FUNCTION_BLOCK TWOCONRINGTOKEN (* Composite Function Block Type *)
  (* Standard: 61499-2 *)
  (* Version 0.2, 2003-12-05, JHC, Rockwell Automation, Renamed from NEWCOMPFB. *)
  (* Version 0.1, 2002-01-08, JHC, Rockwell Automation, Added DLY FB as example. *)
  (* Version 0.0, 2000-05-27, JHC, Rockwell Automation *)
  (* Compiler header: package fb.rt.cs725; *)
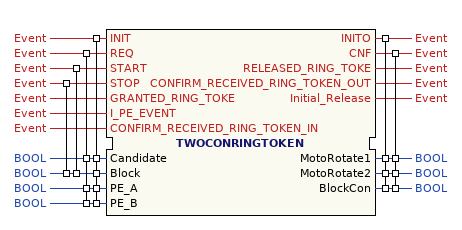
  EVENT_INPUT
    INIT WITH Candidate, Block, PE_A, PE_B; (* Initialization Request *)
    REQ WITH Candidate, PE_A, PE_B; (* Normal Execution Request *)
    START WITH Block;
    STOP WITH Block;
    GRANTED_RING_TOKE;
    I_PE_EVENT;
    CONFIRM_RECEIVED_RING_TOKEN_IN;
  END_EVENT
  EVENT_OUTPUT
    INITO WITH MotoRotate1, MotoRotate2, BlockCon; (* Initialization Confirm *)
    CNF WITH MotoRotate1, MotoRotate2, BlockCon; (* Execution Confirmation *)
    RELEASED_RING_TOKE;
    CONFIRM_RECEIVED_RING_TOKEN_OUT;
    Initial_Release;
  END_EVENT
  VAR_INPUT
    Candidate : BOOL;
    Block : BOOL;
    PE_A : BOOL;
    PE_B : BOOL;
  END_VAR
  VAR_OUTPUT
    MotoRotate1 : BOOL;
    MotoRotate2 : BOOL;
    BlockCon : BOOL;
  END_VAR
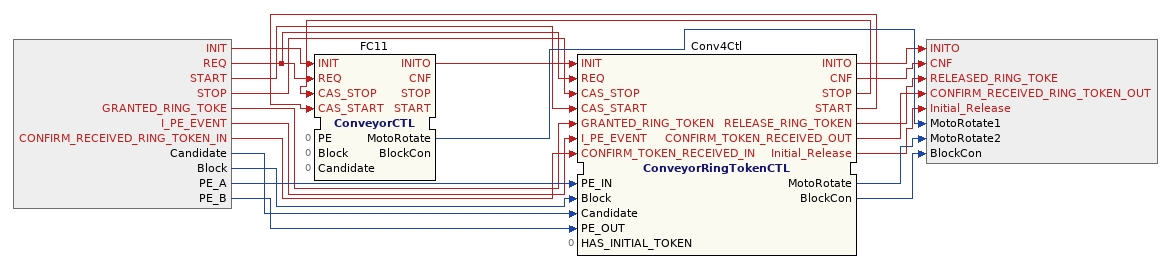
  FBS
    FC11 : ConveyorCTL(Candidate := 0, Block := 0, PE := 0);
    Conv4Ctl : ConveyorRingTokenCTL(HAS_INITIAL_TOKEN := 0);
  END_FBS
  EVENT_CONNECTIONS
    INIT TO FC11.INIT;
    REQ TO FC11.REQ;
    Conv4Ctl.INITO TO INITO;
    Conv4Ctl.CNF TO CNF;
    REQ TO Conv4Ctl.REQ;
    STOP TO Conv4Ctl.CAS_STOP;
    START TO Conv4Ctl.CAS_START;
    Conv4Ctl.STOP TO FC11.CAS_STOP;
    Conv4Ctl.START TO FC11.CAS_START;
    FC11.INITO TO Conv4Ctl.INIT;
    GRANTED_RING_TOKE TO Conv4Ctl.GRANTED_RING_TOKEN;
    Conv4Ctl.RELEASE_RING_TOKEN TO RELEASED_RING_TOKE;
    I_PE_EVENT TO Conv4Ctl.I_PE_EVENT;
    CONFIRM_RECEIVED_RING_TOKEN_IN TO Conv4Ctl.CONFIRM_TOKEN_RECEIVED_IN;
    Conv4Ctl.CONFIRM_TOKEN_RECEIVED_OUT TO CONFIRM_RECEIVED_RING_TOKEN_OUT;
    Conv4Ctl.Initial_Release TO Initial_Release;
  END_CONNECTIONS
  DATA_CONNECTIONS
    Block TO Conv4Ctl.Block;
    Candidate TO Conv4Ctl.Candidate;
    Conv4Ctl.BlockCon TO BlockCon;
    FC11.MotoRotate TO MotoRotate1;
    Conv4Ctl.MotoRotate TO MotoRotate2;
    PE_A TO Conv4Ctl.PE_IN;
    PE_B TO Conv4Ctl.PE_OUT;
  END_CONNECTIONS
END_FUNCTION_BLOCK
